// TIA Portal V19 export
FUNCTION "Burkert_CH_T8691_rev3" : Void   // FC117, STL
{ S7_Optimized_Access := 'TRUE' }
// Data words uses in function
// 
// HMI_CMD, dw X - command word from SCADA
// Bit 0 = auto
// Bit 1 = Manuel deactivate
// Bit 2 = Manuel activate
// Bit 3 = Locate
// Bit 4 = Teach
// Bit 5 = spare
// Bit 6 = spare
// 
// HMI_INFO, dw X - info word to SCADA
// Bit 0  = activated
// Bit 1  = changing
// Bit 2  = faulty 
// Bit 3  = auto_man, Manuel = 1 
// Bit 4  = man_on_off
// Bit 5  = Reset_FB
// Bit 6  = ManualSelected
// Bit 7  = Set_FB
// Bit 8  = Locate Active 
// Bit 9  = spare 
// Bit 10 = spare 
// Bit 11 = spare  
// Bit 12 = spare 
// Bit 13 = spare 
// Bit 14 = fb_error - Alarm feedback error
// Bit 15 = spare 
// 
// OperationalState: 0=Initialisation,1=Teach function,2=Normal Operation,3=Safety 
// end position,4=MANUAL Operation State,5= Teach in Operation
// stored: AutoNumber false
   VAR_INPUT
      Addr : Int;   // First Byte address of 4 byte address space
      Locate : Bool;   // Rapid Flash LED's
      Activate : Bool;   // Activate pilot valve
   END_VAR
   VAR_OUTPUT
      ValvePosition : Real;   // 0-100%
      OperationState : Byte;   // See block comment
      POS2 : Bool;   // True = process valve is in end position defined by activated pilot valve.
      POS1 : Bool;   // True = process valve is in end position defined by deactivated pilot valve.
      O_DI4 : Bool;   // Output signal status Pin 4
      O_DI2 : Bool;   // Output signal status Pin 2
      Teach : Bool;   // Teach output for command bit
   END_VAR
   VAR_IN_OUT
      itemInfo : "ItemInfo_UDT";
      itemCommand : "ItemCommand_UDT";
      EndPositionClose : Bool;   // True = Process Valve is closed.
      EndPositionOpen : Bool;   // True = Process Valve is open.
      NumarState : Byte;   // 0=diagPassive,1=diagActive,2=MaintenanceRequired,3=OutOfSpec,4=warn,5=error
      O_DA : Bool;   // Output device recognised
      O_DE : Bool;   // Output device error event has appeared
      O_PQ : Bool;   // Output port qualifer proces data valid
   END_VAR
   VAR_TEMP
      TW_Flag : Word;
      output : Bool;
   END_VAR
BEGIN

NETWORK
TITLE = info to scada, free
// L     #HMI_INFO
// Get first byte address
      L     #Addr;
      SLW   3;
      LAR1;
// **************  Inputs *******************
// Valve Position
      L     ID [AR1, P#0.0];
      T     #ValvePosition;

// Namur State
      L     IB [AR1, P#4.0];
      T     #NumarState;

// Operation State
      L     IB [AR1, P#5.0];
      T     #OperationState;

// POS2
      L     IB [AR1, P#6.0];
      T     #TW_Flag;
      L     8;
      AW;
      L     8;
      ==I;
      =     #POS2;


// POS1
      L     IB [AR1, P#6.0];
      T     #TW_Flag;
      L     4;
      AW;
      L     4;
      ==I;
      =     #POS1;
// Valve Closed
      L     IB [AR1, P#6.0];
      T     #TW_Flag;
      L     1;
      AW;
      L     1;
      ==I;
      =     #EndPositionClose;


// Valve Opened
      L     IB [AR1, P#6.0];
      T     #TW_Flag;
      L     2;
      AW;
      L     2;
      ==I;
      =     #EndPositionOpen;


// PQI

      L     IB [AR1, P#8.0];
      T     #TW_Flag;

      L     #TW_Flag;
      L     1;
      AW;
      L     1;
      ==I;
      =     #O_DI4;



      L     #TW_Flag;
      L     2;
      AW;
      L     2;
      ==I;
      =     #O_DI2;

      L     #TW_Flag;
      L     32;
      AW;
      L     32;
      ==I;
      =     #O_DA;

      L     #TW_Flag;
      L     64;
      AW;
      L     64;
      ==I;
      =     #O_DE;


      L     #TW_Flag;
      L     128;
      AW;
      L     128;
      ==I;
      =     #O_PQ;

// *** Valve Fault Detected ***
      L     #NumarState;
      L     1;
      >I;
      O;
      A     #O_DE;
      O;
      AN    #O_DA;
      AN    #O_DE;
      AN    #O_PQ;
      =     #itemInfo.fb_error;
//
// Valve Control

      AN    #itemInfo.auto_man;  // IF AUTO
      A     #Activate;  // AND ProcessReq
      O(;
      A     #itemInfo.auto_man;  // IF Manuel
      A     #itemInfo.man_on_off;  // Manuel on/off
      );
      =     Q [AR1, P#0.0];  // Set/reset Output
      =     #output;

// Locate

      A     #itemCommand.Locate;
      A     #itemInfo.LocateActive;
      R     Q [AR1, P#0.1];
      R     #itemCommand.Locate;


      A     #itemCommand.Locate;
      AN    #itemInfo.LocateActive;
      S     Q [AR1, P#0.1];
      R     #itemCommand.Locate;


//****************** Outputs ************

      L     QB [AR1, P#0.0];
      T     QB [AR1, P#0.0];

// Teach

      A     #itemCommand.Teach;
      =     #Teach;



NETWORK
TITLE = SCADA INFO & command
      AN    #itemCommand.Auto;
      AN    #itemCommand.Locate;
      AN    #itemCommand.Man_Act;
      AN    #itemCommand.Man_DeAct;
      AN    #itemCommand.Teach;
      AN    #itemCommand.SpareBool;
      AN    #itemCommand.SpareBool_1;
      AN    #itemCommand.SpareBool_2;
      AN    #itemCommand.SpareBool_3;
      AN    #itemCommand.SpareBool_4;
      AN    #itemCommand.SpareBool_5;
      AN    #itemCommand.SpareBool_6;
      AN    #itemCommand.SpareBool_7;
      AN    #itemCommand.SV_2SelectionBit;
      AN    #itemCommand.SV_3SelectionBit;
      AN    #itemCommand.SpareBool_10;
      JC    INFO;  // if commamd bits = 0 then no commands


      A     #itemCommand.Auto;
      R     #itemInfo.auto_man;
      JC    clea;

      A     #itemCommand.Man_DeAct;
      S     #itemInfo.auto_man;
      R     #itemInfo.man_on_off;
      JC    clea;

      A     #itemCommand.Man_Act;
      S     #itemInfo.auto_man;
      S     #itemInfo.man_on_off;
      JC    clea;
// Clear itemCommand word
clea: SET;
      R     #itemCommand.Auto;
      R     #itemCommand.Locate;
      R     #itemCommand.Man_Act;
      R     #itemCommand.Man_DeAct;
      R     #itemCommand.Teach;
      R     #itemCommand.SpareBool;
      R     #itemCommand.SpareBool_1;
      R     #itemCommand.SpareBool_2;
      R     #itemCommand.SpareBool_3;
      R     #itemCommand.SpareBool_4;
      R     #itemCommand.SpareBool_5;
      R     #itemCommand.SpareBool_6;
      R     #itemCommand.SpareBool_7;
      R     #itemCommand.SV_2SelectionBit;
      R     #itemCommand.SV_3SelectionBit;
      R     #itemCommand.SpareBool_10;
//clear command word


//;=========================== Scada info ================================
INFO: A     #itemInfo.fb_error;  // feedback error
      =     #itemInfo.faulty;
      A     #itemInfo.auto_man;
      =     #itemInfo.ManualSelected;  //Show Manual selected on SCADA
      A     #EndPositionClose;
      =     #itemInfo.Reset_FB;  //Show Reset FB in "Item Info & Operation" popup
      A     #EndPositionOpen;
      =     #itemInfo.Set_FB;  //Show Set FB in "Item Info & Operation" popup
      A     Q [AR1, P#0.1];
      =     #itemInfo.LocateActive;


//;                     // ================================
//;                     // = SET FB , SET/RES FB =
      A     #output;  // IF Output
      A     #EndPositionOpen;  // AND SetFB
      JC    ACT;  // Goto Activated

      A     #output;  // IF Output
      AN    #EndPositionClose;  // AND NOT SetFB
      JC    CHAN;  // Goto Changing

      JU    DEAC;
//;                     // ================================
//;                     // ================================
DEAC: R     #itemInfo.activated;  // Update = deactivated
      R     #itemInfo.changing;
      JU    NEX4;  //NEXT;
//;                     // ================================
CHAN: R     #itemInfo.activated;  // Update = activated
      S     #itemInfo.changing;
      JU    NEX4;  //NEXT;
//;                     // ================================
ACT:  S     #itemInfo.activated;  // Update = activated
      R     #itemInfo.changing;
      JU    NEX4;  //NEXT;
//;                     // ================================
NEX4: NOP   0;


END_FUNCTION
